(* Logix 5000 project; controller MetsoFilter vendor 1 type 14 code 106 rev 32.11; software revision 32.00; part 3 of 4 *)
(* tags used below, declared in another part *)
   AlarmHornPulser : BOOL;   // Pulse Horn during a new alarm
   AlarmReset : BOOL;   // Alarm Rest Relay
   ALM_W2 : DINT;   // Alarms to HMI, Word #2
   AlwaysOff : BOOL;   // Always Off Bit
   AS_AirDry : BOOL;   // Auto Sequence, Air Dry
   AS_ClothVibWash : BOOL;   // Auto Sequence Vibrate & Wash Cloth
   AS_ClothVibWash_T : TIMER;   // Auto Sequence Vibrate & Wash Cloth Timer
   AS_Drain : BOOL;   // Auto Sequence, Drain
   AS_HPC_Open_V1_T : TIMER;   // Auto Sequence, Open Slurry Valve V1 Timer
   AS_LowFeedWeight : BOOL;   // Auto Sequence, Low Feed Weight, Enable Retry
   AS_LowPressClose : BOOL;   // Auto Sequence, Close Press at Low Pressure
   AS_MembComp : BOOL;   // Auto Sequence, Membrane Compress
   AS_MembComp_Ena : BOOL;   // Auto Sequence, Enable Membrane Compress When in Auto Run
   AS_TopBlow_Wat : BOOL;   // Auto Sequence, Top Blow Water
   AS_TopBlowAir1 : BOOL;   // Auto Sequence, Top Blow Air #1
   AS_TopBlowAir1_T : TIMER;   // Auto Sequence, Top Blow Air #1 Timer
   AS_TopBlowAir2 : BOOL;   // Auto Sequence, Top Blow Air #2
   AS_TopBlowAir2_T : TIMER;   // Auto Sequence, Top Blow Air #2 Timer
   AS_VibrateCloth : BOOL;   // Auto Sequence Vibrate Cloth
   AS_VibrateCloth_T : TIMER;   // Auto Sequence Vibrate Cloth Timer
   Auto_Run : BOOL;   // Run the Next Step of the Auto Sequence
   AutoSeqStarted : BOOL;   // Auto Sequence Started
   ClothDamaged_T : TIMER;   // Dammaged Cloth Detection Switch On Plus Time
   Colon_STR : STRING;   // Constant Colon String = ":"
   Dash_STR : STRING;   // Constant Dash String = "-"
   DateTimeArray : DINT[7];
   Day_STR : STRING;   // Day String(1-31)
   DD_Cycle_1 : Status_Cycle;   // Cycle 1 At Left Side Of Statistics Screen
   DD_Cycle_2 : Status_Cycle;   // Cycle 2
   DD_Cycle_3 : Status_Cycle;   // Cycle 3
   DD_Cycle_4 : Status_Cycle;   // Cycle 4
   DD_Cycle_5 : Status_Cycle;   // Cycle 5
   DD_Cycle_6 : Status_Cycle;   // Cycle 6
   DD_Cycle_7_Now : Status_Cycle;   // Cycle 7, Now being Updated @ Right Side of Statistics Screen
   DD_CyclesLeft : DINT;   // To HMI, Cycles Left Before Servicing
   DD_CycleTime : DINT;   // To HMI, Current Cycle time
   DD_Date_STR : STRING;   // Date String - YYYY-MM-DD
   DD_Day_1 : Status_Day;   // Status Day 1 At Left Side of Statistics Screen
   DD_Day_2 : Status_Day;   // Status Day 2
   DD_Day_3 : Status_Day;   // Status Day 3
   DD_Day_4 : Status_Day;   // Status Day 4
   DD_Day_5 : Status_Day;   // Status Day 5
   DD_Day_6 : Status_Day;   // Status Day 6
   DD_Day_7_Now : Status_Day;   // Status Day 7, Now Being Updated @ Right Side of Statistics Screen
   DD_LastResetDate_STR : DINT;   // On Statistics Screen, Date when last reset performed
   DD_PressWeight : DINT;   // Press Weight from Analog Input Data Display
   DD_Shift3_Start : DINT;   // To HMI, Shift 3 Start Hour
   DD_Time_STR : STRING;   // Time String = HH:MM
   DD_TotalCycles : DINT;   // To HMI, Total Cycles Performed, since last Reset
   DD_TotalTons : DINT;   // To HMI, Total Tons Pressed from Last Reset
   DE_ServiceCycles : DINT;   // Special Screen, Service Cycles for Maintenance Data Entry
   DE_Shift1_Start : DINT;   // Special Screen, Shift1 Start Hour, Data Entry
   DE_Shift2_Start : DINT;   // Special Screen, Shift 2 Start Data Entry
   DSH1 : BOOL;   // Dammaged Cloth Detection Switch
   DummyOutput : BOOL;   // Dummy Output for Temporary outputs File
   GSC11 : BOOL;   // Upper Hatch is Closed Proximity Switch
   GSC9 : BOOL;   // Lower Hatch is Closed Proximity Switch
   GSO10 : BOOL;   // Lower Hatch is Open Proximity Switch
   GSO12 : BOOL;   // Upper Hatch is Open Proximity Switch
   H1b : BOOL;   // Hydraulic Valve, Main Drainage
   H2a : BOOL;   // Hydraulic Valve, High Pressure Drainage
   H2b : BOOL;   // Hydraulic Valve, High Pressure Close
   H3a : BOOL;   // Hydraulic Valve, Press Close
   H3b : BOOL;   // Hydraulic Valve, Press Open
   H4a : BOOL;   // Hydraulic Valve, Raise (Open) Lower Hatch
   H4b : BOOL;   // Hydraulic Valve, Lower (Close) Lower Hatch
   H5a : BOOL;   // Hydraulic Valve, Raise (Open) Upper Hatch
   H5b : BOOL;   // Hydraulic Valve, Lower (Close) Upper Hatch
   HornPulseDuration_T : TIMER;   // Pulse Horn Duration Timer
   HornPulseOff_T : TIMER;   // Pulse Horn Off Timer
   HornPulses_C : COUNTER;   // Number of times horn pusles for new alarm
   Hour_STR : STRING;   // Hour String(0-23)
   M_HPP_Run : BOOL;   // High Pressure Pump Run Output Bit
   M_HPP_Running : BOOL;   // High Pressure Pump is Running
   M_LPP_Run : BOOL;   // Low Pressure Pump Run Output Bit
   M_Vibrator_Run : BOOL;   // Vibrator Motor Run Output
   M_Vibrator_Run_T : TIMER;   // Vibrator Motor Run Output On Plus Time
   M_Vibrator_Running : BOOL;   // Vibrator Motor Running Input
   MAN_Vibrate : BOOL;   // Manual Vibrate Flip Flop
   Manual_ON : BOOL;   // Manual On Mode
   MAS_CloseHatch : BOOL;   // Manual / Auto Close Hatch
   MAS_CloseUpperHatch_T : TIMER;   // Manual / Auto Close Upper Hatch Delay Timer
   MAS_OpenHatch : BOOL;   // Manual / Auto Open Hatch
   MAS_OpenLowerHatch_T : TIMER;   // Manual / Auto Open Hatch, Delay Lower Hatch Open
   Minute_STR : STRING;   // Minute String(0-59)
   Month_STR : STRING;   // Month String(1-12)
   NewAlarm_OS : BOOL;   // A New Alarm Has Occured
   NewAlarm_PulseHorn : BOOL;   // A New Alarm has Occured, pulse the Horn
   NumberOfAlarms : DINT;   // Number of Active Alarms
   NumberOfAlarms_LS : DINT;   // Number of Active Alarms Last Scan, Detect New Alarm
   OneThirdAir1Preset : DINT;   // 1/3 Top Blow Air 1 time
   OneThirdAir2Preset : DINT;   // 1/3 Top Blow Air 2 time
   PB_AlarmAck : BOOL;   // Alarm Acknowledge Pushbutton
   PB_AlarmReset : BOOL;   // Alarm Reset Pushbutton
   PB_ResetSpecial : BOOL;   // Reset Pushbutton on the Specal Screen, Reset Total Cycles & Weight
   S_AS_DoneOS : BOOL;   // Statistics, Automatic Sequence Normally Done or Abnormally Stopped One Shot
   S_AS_DoneOSB : BOOL;   // Statistics, Automatic Sequence Done One Shot
   S_AS_StartOS : BOOL;   // Statistics, Automatic Sequence Started One Shot
   S_AS_StartOSB : BOOL;   // Statistics, Automatic Sequence Started One Shot
   S_CloseHatchOSB : BOOL;   // Statistics, Hatch Starting to Close, One Shot
   S_CycleTimer : TIMER;   // Statistics, Cycle Time Timer
   S_DryingTimer : TIMER;   // Statistics, Drying Time Timer
   S_NewDay : BOOL;   // Statistics, Midnight & No Sequence Running, Update Days
   S_OpenHatchOSB : BOOL;   // Statistics, Hatch Starting to Open, One Shot
   S_PressWeightTons : REAL;   // Statistics, Weight in Tons Just Pressed
   S_PumpTimer : TIMER;   // Statistics, Pump Time Timer
   S_Shift1 : BOOL;   // Statistics, Shift 1 in Progress
   S_Shift1_OSB : BOOL;   // Statistics, Start of Shift 1 One shot
   S_Shift2 : BOOL;   // Statistics, Shift 2 in Progress
   S_Shift2_OSB : BOOL;   // Statistics, Start of Shift 2 One shot
   S_Shift3 : BOOL;   // Statistics, Shift 3 in Progress
   S_Shift3_OSB : BOOL;   // Statistics, Start of Shift 3 One shot
   S_TempDINT : DINT;   // Statistics, Tempory Holding DINT
   S_WeightHatchOpen : DINT;   // Statistics, Weight of Press just as hatches Open
   S_ZeroHour_Latch : BOOL;   // Zero Hour Latch, wait for current sequence to finish, if running
   S_ZeroHour_OSB : BOOL;   // Hour = Zero, New Day One Shot
   TwoThirdsAir1Preset : DINT;   // 2/3 Top Blow Air 1 time
   TwoThirdsAir2Preset : DINT;   // 2/3 Top Blow Air 2 time
   Year_STR : STRING;   // Year String
   YV1 : BOOL;   // Valve #1, Slurry Supply, Open Output Bit
   YV10 : BOOL;   // Valve #10, Membrane Drain, Normally Open, Energize to Close, Output Bit
   YV3 : BOOL;   // Valve #3, Filtrate, Open Output Bit
   YV4 : BOOL;   // Valve #4, Slurry Return, Open Output Bit
   YV5 : BOOL;   // Valve #5, Drying Air, Open Output Bit
   YV6 : BOOL;   // Valve #6, Top Blow Air, Open Output Bit
   YV7 : BOOL;   // Valve #7, Membrane Air, Open Output Bit
   YV8 : BOOL;   // Valve #8, Top Blow Water, Open Output Bit
   YV9 : BOOL;   // Valve #9, Wash Water, Open Ouput Bit
   Zero_STR : STRING;   // Constant String= "0" Pad Values <10 0-9 -> 00-09
(* MainProgram, continued *)

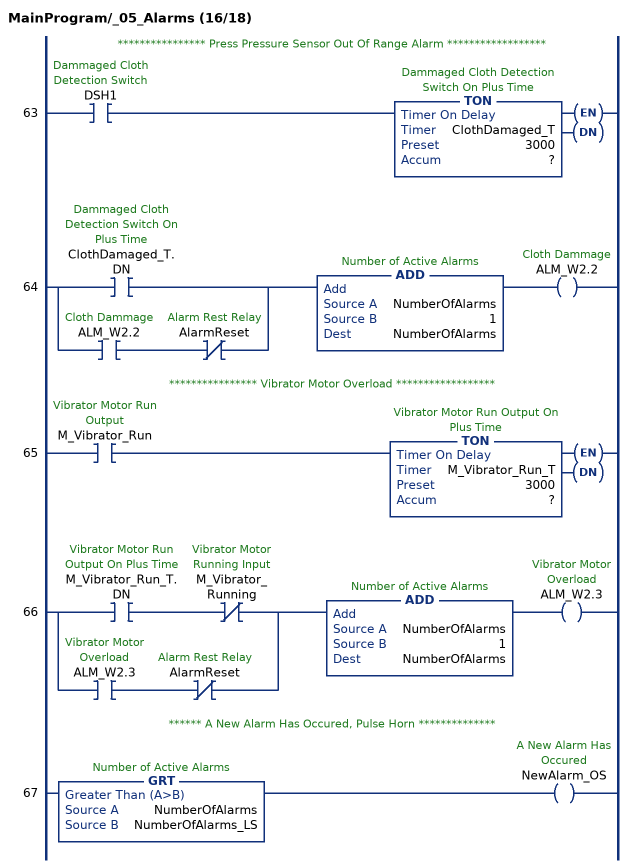
   [picture p48: MainProgram/_05_Alarms rungs 63-67]
   // **************** Press Pressure Sensor Out Of Range Alarm ******************
   63: XIC(DSH1)TON(ClothDamaged_T,?,?);
   64: [XIC(ClothDamaged_T.DN) ,XIC(ALM_W2.2) XIO(AlarmReset) ]ADD(NumberOfAlarms,1,NumberOfAlarms)OTE(ALM_W2.2);
   // **************** Vibrator Motor Overload ******************
   65: XIC(M_Vibrator_Run)TON(M_Vibrator_Run_T,?,?);
   66: [XIC(M_Vibrator_Run_T.DN) XIO(M_Vibrator_Running) ,XIC(ALM_W2.3) XIO(AlarmReset) ]ADD(NumberOfAlarms,1,NumberOfAlarms)OTE(ALM_W2.3);
   // ****** A New Alarm Has Occured, Pulse Horn **************
   67: GRT(NumberOfAlarms,NumberOfAlarms_LS)OTE(NewAlarm_OS);
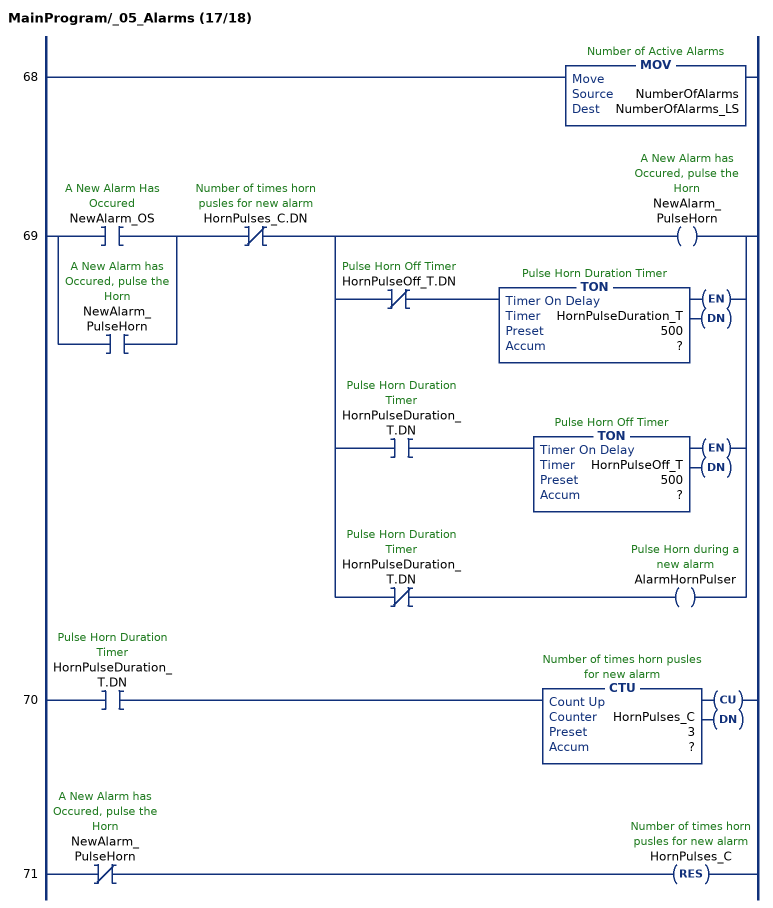
   68: MOV(NumberOfAlarms,NumberOfAlarms_LS);
   69: [XIC(NewAlarm_OS) ,XIC(NewAlarm_PulseHorn) ]XIO(HornPulses_C.DN)[OTE(NewAlarm_PulseHorn) ,XIO(HornPulseOff_T.DN) TON(HornPulseDuration_T,?,?) ,XIC(HornPulseDuration_T.DN) TON(HornPulseOff_T,?,?) ,XIO(HornPulseDuration_T.DN) OTE(AlarmHornPulser) ];
   70: XIC(HornPulseDuration_T.DN)CTU(HornPulses_C,?,?);
   71: XIO(NewAlarm_PulseHorn)RES(HornPulses_C);
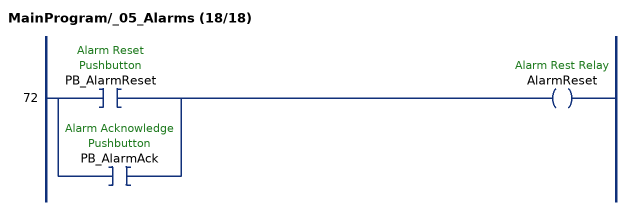
   72: [XIC(PB_AlarmReset) ,XIC(PB_AlarmAck) ]OTE(AlarmReset);
END_ROUTINE

ROUTINE _06_Output_Bits   (* ladder *)
// Set the Output Bits per Manual and Automatic Logic
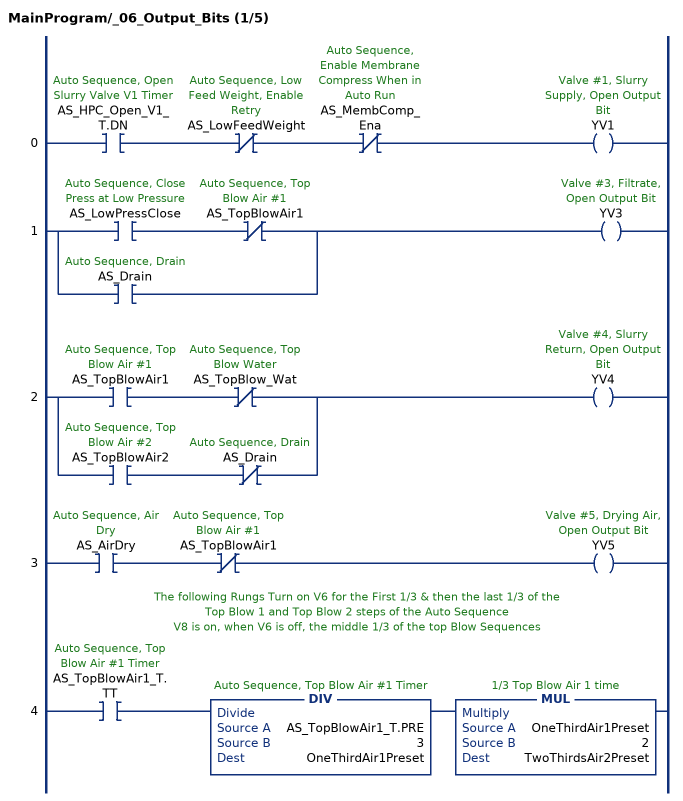
   0: XIC(AS_HPC_Open_V1_T.DN)XIO(AS_LowFeedWeight)XIO(AS_MembComp_Ena)OTE(YV1);
   1: [XIC(AS_LowPressClose) XIO(AS_TopBlowAir1) ,XIC(AS_Drain) ]OTE(YV3);
   2: [XIC(AS_TopBlowAir1) XIO(AS_TopBlow_Wat) ,XIC(AS_TopBlowAir2) XIO(AS_Drain) ]OTE(YV4);
   3: XIC(AS_AirDry)XIO(AS_TopBlowAir1)OTE(YV5);
   // The following Rungs Turn on V6 for the First 1/3 & then the last 1/3 of the
   // Top Blow 1 and Top Blow 2 steps of the Auto Sequence
   // V8 is on, when V6 is off, the middle 1/3 of the top Blow Sequences
   4: XIC(AS_TopBlowAir1_T.TT)DIV(AS_TopBlowAir1_T.PRE,3,OneThirdAir1Preset)MUL(OneThirdAir1Preset,2,TwoThirdsAir2Preset);
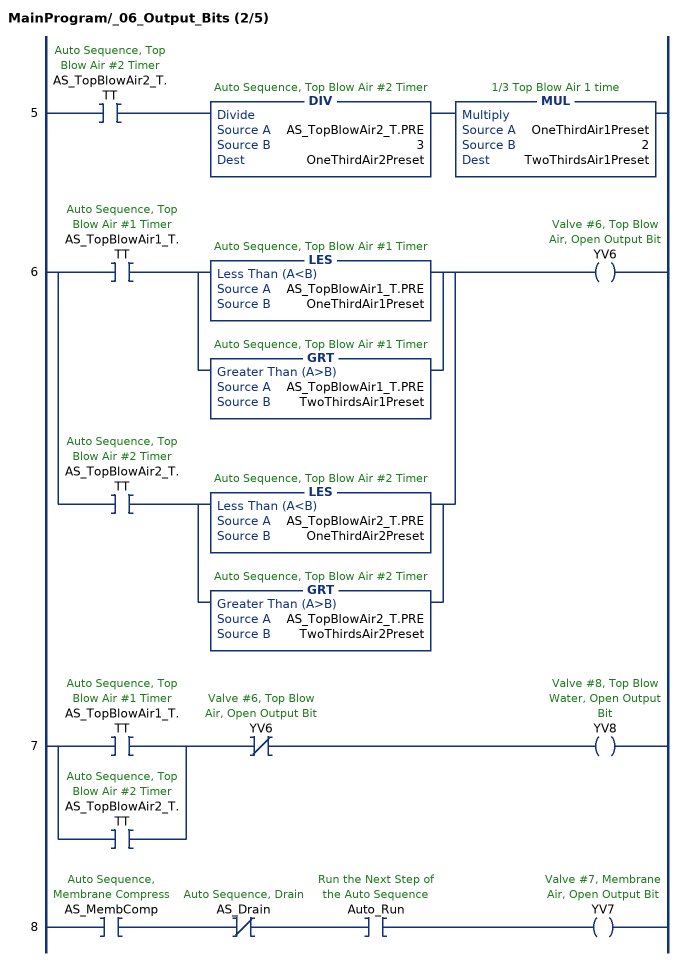
   5: XIC(AS_TopBlowAir2_T.TT)DIV(AS_TopBlowAir2_T.PRE,3,OneThirdAir2Preset)MUL(OneThirdAir1Preset,2,TwoThirdsAir1Preset);
   6: [XIC(AS_TopBlowAir1_T.TT) [LES(AS_TopBlowAir1_T.PRE,OneThirdAir1Preset) ,GRT(AS_TopBlowAir1_T.PRE,TwoThirdsAir1Preset) ] ,XIC(AS_TopBlowAir2_T.TT) [LES(AS_TopBlowAir2_T.PRE,OneThirdAir2Preset) ,GRT(AS_TopBlowAir2_T.PRE,TwoThirdsAir2Preset) ] ]OTE(YV6);
   7: [XIC(AS_TopBlowAir1_T.TT) ,XIC(AS_TopBlowAir2_T.TT) ]XIO(YV6)OTE(YV8);
   8: XIC(AS_MembComp)XIO(AS_Drain)XIC(Auto_Run)OTE(YV7);
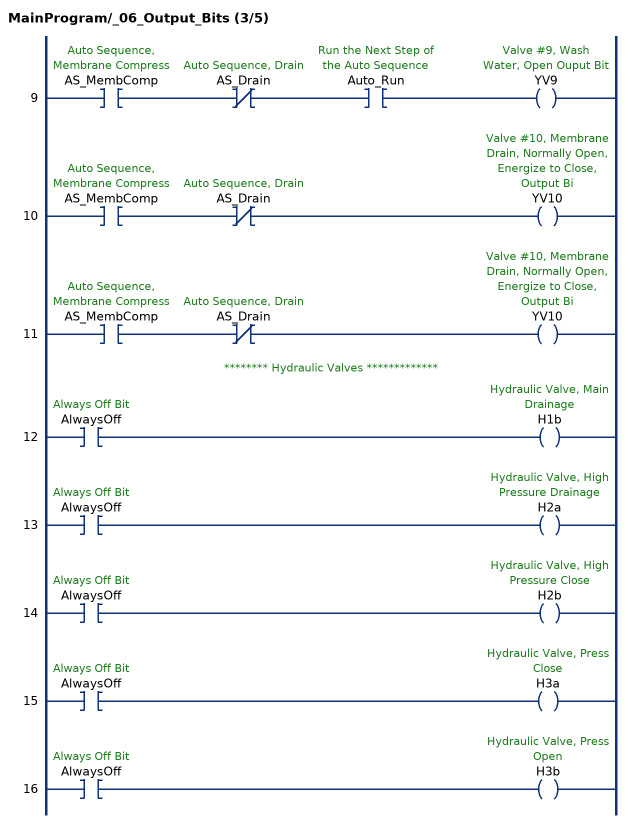
   9: XIC(AS_MembComp)XIO(AS_Drain)XIC(Auto_Run)OTE(YV9);
   10: XIC(AS_MembComp)XIO(AS_Drain)OTE(YV10);
   11: XIC(AS_MembComp)XIO(AS_Drain)OTE(YV10);
   // ******** Hydraulic Valves *************
   12: XIC(AlwaysOff)OTE(H1b);
   13: XIC(AlwaysOff)OTE(H2a);
   14: XIC(AlwaysOff)OTE(H2b);
   15: XIC(AlwaysOff)OTE(H3a);
   16: XIC(AlwaysOff)OTE(H3b);
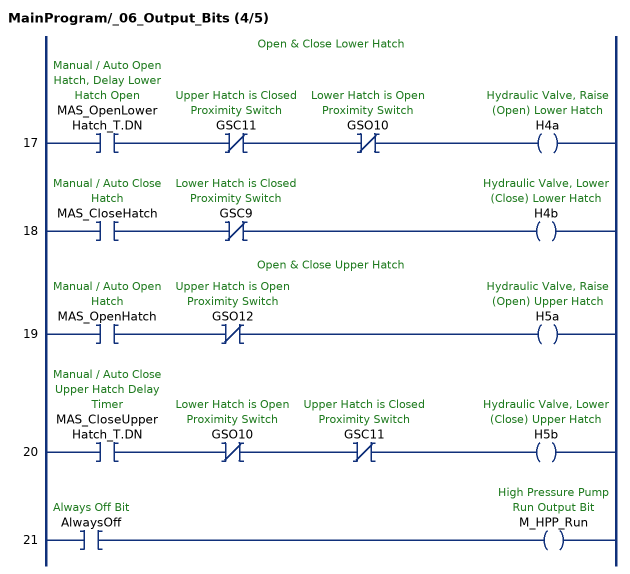
   // Open & Close Lower Hatch
   17: XIC(MAS_OpenLowerHatch_T.DN)XIO(GSC11)XIO(GSO10)OTE(H4a);
   18: XIC(MAS_CloseHatch)XIO(GSC9)OTE(H4b);
   // Open & Close Upper Hatch
   19: XIC(MAS_OpenHatch)XIO(GSO12)OTE(H5a);
   20: XIC(MAS_CloseUpperHatch_T.DN)XIO(GSO10)XIO(GSC11)OTE(H5b);
   21: XIC(AlwaysOff)OTE(M_HPP_Run);
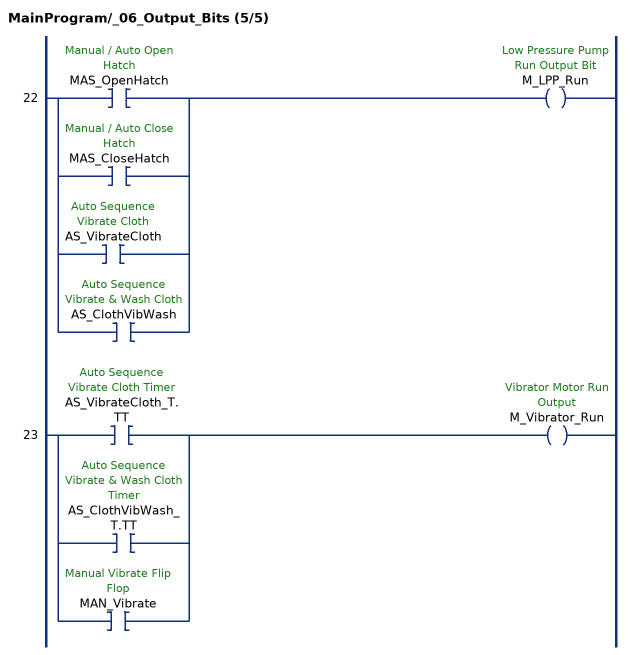
   22: [XIC(MAS_OpenHatch) ,XIC(MAS_CloseHatch) ,XIC(AS_VibrateCloth) ,XIC(AS_ClothVibWash) ]OTE(M_LPP_Run);
   23: [XIC(AS_VibrateCloth_T.TT) ,XIC(AS_ClothVibWash_T.TT) ,XIC(MAN_Vibrate) ]OTE(M_Vibrator_Run);
END_ROUTINE

ROUTINE _07_MapOutputs   (* ladder *)
// Map Output Bits to PLC Outputs
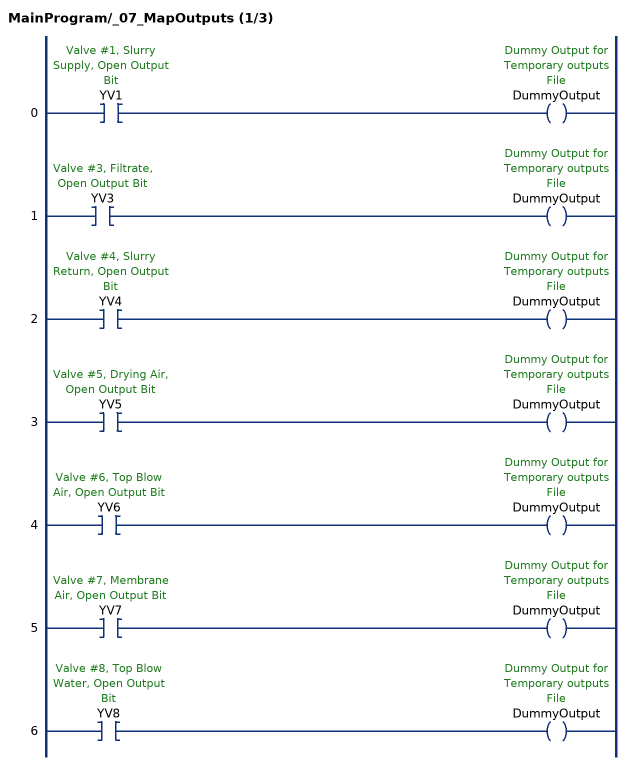
   0: XIC(YV1)OTE(DummyOutput);
   1: XIC(YV3)OTE(DummyOutput);
   2: XIC(YV4)OTE(DummyOutput);
   3: XIC(YV5)OTE(DummyOutput);
   4: XIC(YV6)OTE(DummyOutput);
   5: XIC(YV7)OTE(DummyOutput);
   6: XIC(YV8)OTE(DummyOutput);
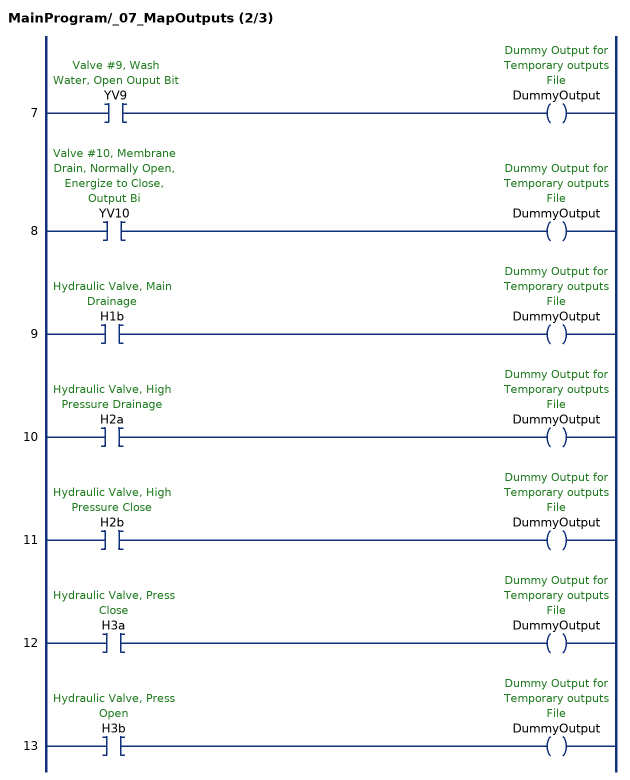
   7: XIC(YV9)OTE(DummyOutput);
   8: XIC(YV10)OTE(DummyOutput);
   9: XIC(H1b)OTE(DummyOutput);
   10: XIC(H2a)OTE(DummyOutput);
   11: XIC(H2b)OTE(DummyOutput);
   12: XIC(H3a)OTE(DummyOutput);
   13: XIC(H3b)OTE(DummyOutput);
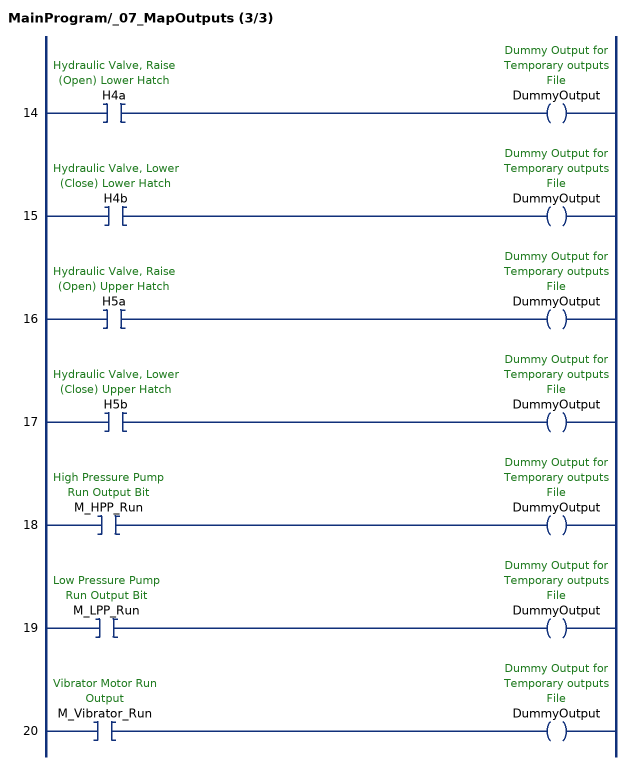
   14: XIC(H4a)OTE(DummyOutput);
   15: XIC(H4b)OTE(DummyOutput);
   16: XIC(H5a)OTE(DummyOutput);
   17: XIC(H5b)OTE(DummyOutput);
   18: XIC(M_HPP_Run)OTE(DummyOutput);
   19: XIC(M_LPP_Run)OTE(DummyOutput);
   20: XIC(M_Vibrator_Run)OTE(DummyOutput);
END_ROUTINE

ROUTINE _08_Statistics   (* ladder *)
// Track Last 7 Days & Cycles
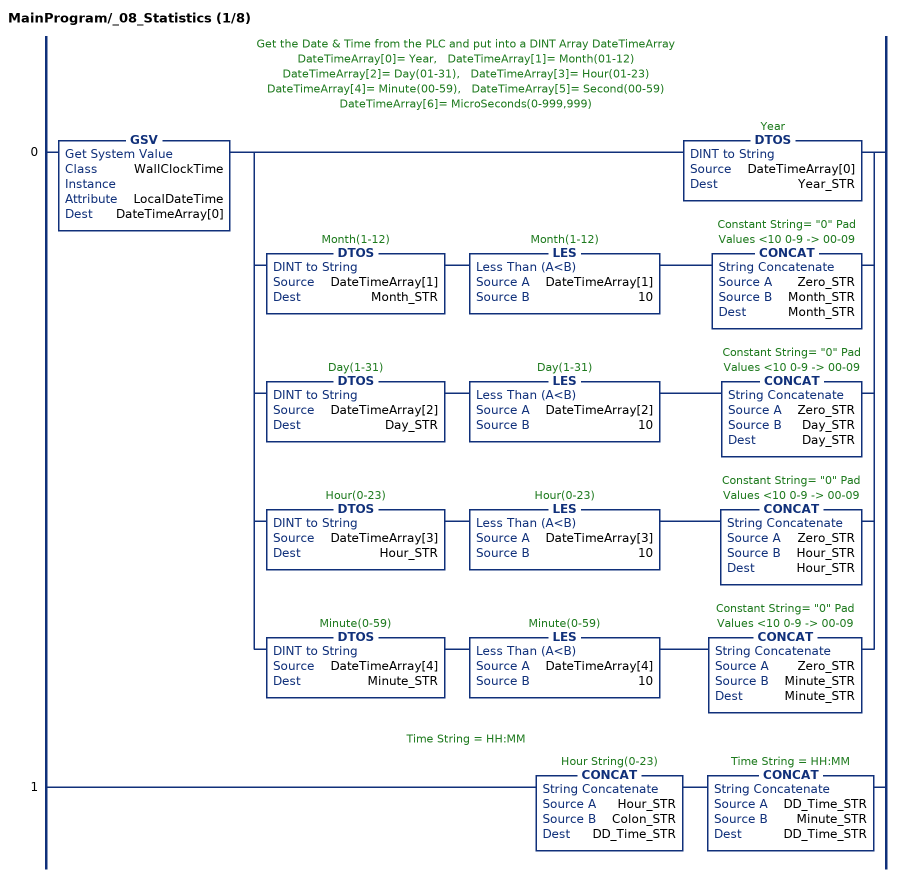
   // Get the Date & Time from the PLC and put into a DINT Array DateTimeArray
   // DateTimeArray[0]= Year,   DateTimeArray[1]= Month(01-12)
   // DateTimeArray[2]= Day(01-31),   DateTimeArray[3]= Hour(01-23)
   // DateTimeArray[4]= Minute(00-59),   DateTimeArray[5]= Second(00-59)
   // DateTimeArray[6]= MicroSeconds(0-999,999)
   0: GSV(WallClockTime,,LocalDateTime,DateTimeArray[0])[DTOS(DateTimeArray[0],Year_STR) ,DTOS(DateTimeArray[1],Month_STR) LES(DateTimeArray[1],10) CONCAT(Zero_STR,Month_STR,Month_STR) ,DTOS(DateTimeArray[2],Day_STR) LES(DateTimeArray[2],10) CONCAT(Zero_STR,Day_STR,Day_STR) ,DTOS(DateTimeArray[3],Hour_STR) LES(DateTimeArray[3],10) CONCAT(Zero_STR,Hour_STR,Hour_STR) ,DTOS(DateTimeArray[4],Minute_STR) LES(DateTimeArray[4],10) CONCAT(Zero_STR,Minute_STR,Minute_STR) ];
   // Time String = HH:MM
   1: CONCAT(Hour_STR,Colon_STR,DD_Time_STR)CONCAT(DD_Time_STR,Minute_STR,DD_Time_STR);
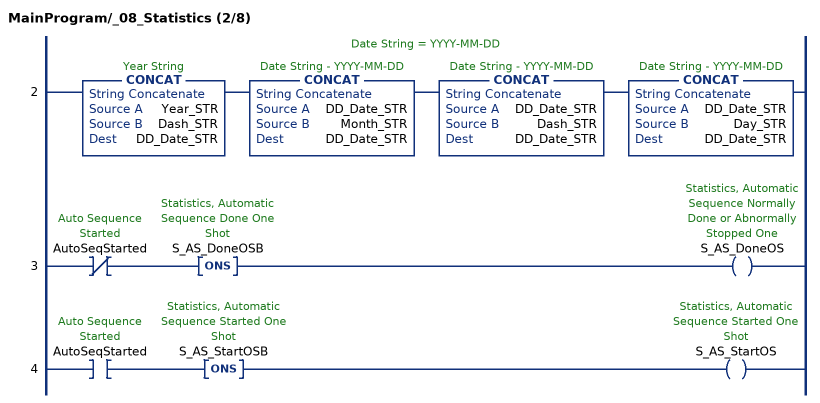
   // Date String = YYYY-MM-DD
   2: CONCAT(Year_STR,Dash_STR,DD_Date_STR)CONCAT(DD_Date_STR,Month_STR,DD_Date_STR)CONCAT(DD_Date_STR,Dash_STR,DD_Date_STR)CONCAT(DD_Date_STR,Day_STR,DD_Date_STR);
   3: XIO(AutoSeqStarted)ONS(S_AS_DoneOSB)OTE(S_AS_DoneOS);
   4: XIC(AutoSeqStarted)ONS(S_AS_StartOSB)OTE(S_AS_StartOS);
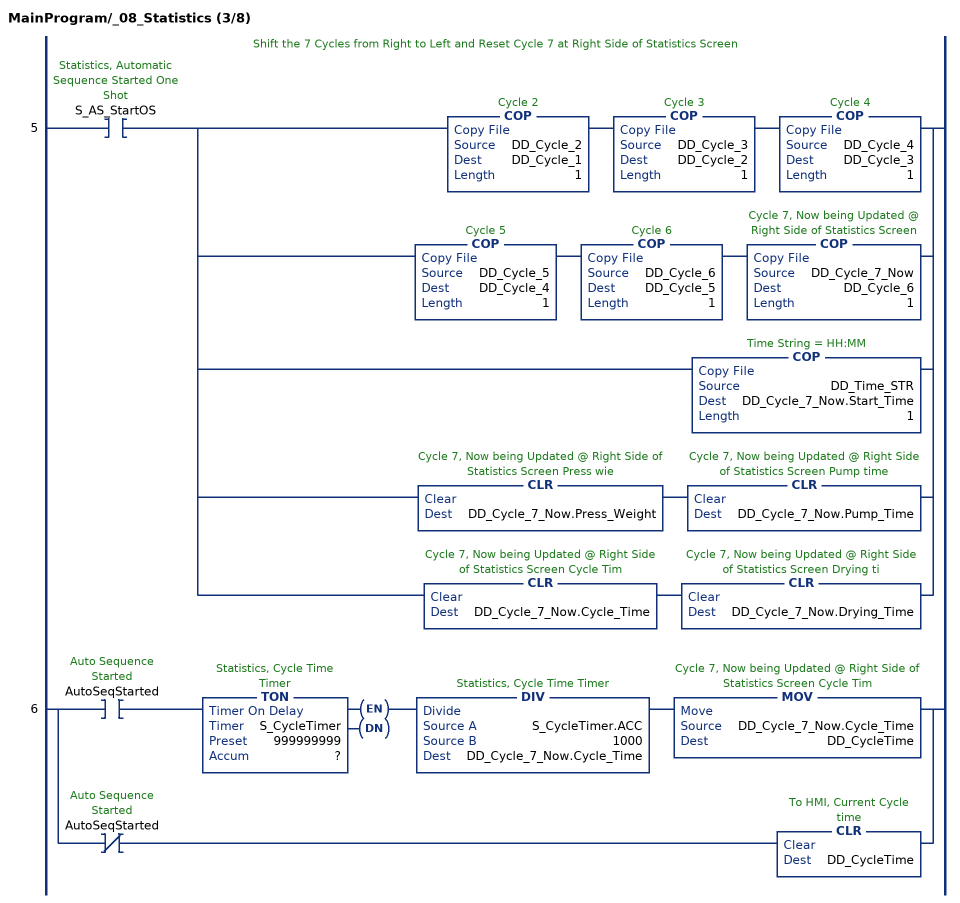
   // Shift the 7 Cycles from Right to Left and Reset Cycle 7 at Right Side of Statistics Screen
   5: XIC(S_AS_StartOS)[COP(DD_Cycle_2,DD_Cycle_1,1) COP(DD_Cycle_3,DD_Cycle_2,1) COP(DD_Cycle_4,DD_Cycle_3,1) ,COP(DD_Cycle_5,DD_Cycle_4,1) COP(DD_Cycle_6,DD_Cycle_5,1) COP(DD_Cycle_7_Now,DD_Cycle_6,1) ,COP(DD_Time_STR,DD_Cycle_7_Now.Start_Time,1) ,CLR(DD_Cycle_7_Now.Press_Weight) CLR(DD_Cycle_7_Now.Pump_Time) ,CLR(DD_Cycle_7_Now.Cycle_Time) CLR(DD_Cycle_7_Now.Drying_Time) ];
   6: [XIC(AutoSeqStarted) TON(S_CycleTimer,?,?) DIV(S_CycleTimer.ACC,1000,DD_Cycle_7_Now.Cycle_Time) MOV(DD_Cycle_7_Now.Cycle_Time,DD_CycleTime) ,XIO(AutoSeqStarted) CLR(DD_CycleTime) ];
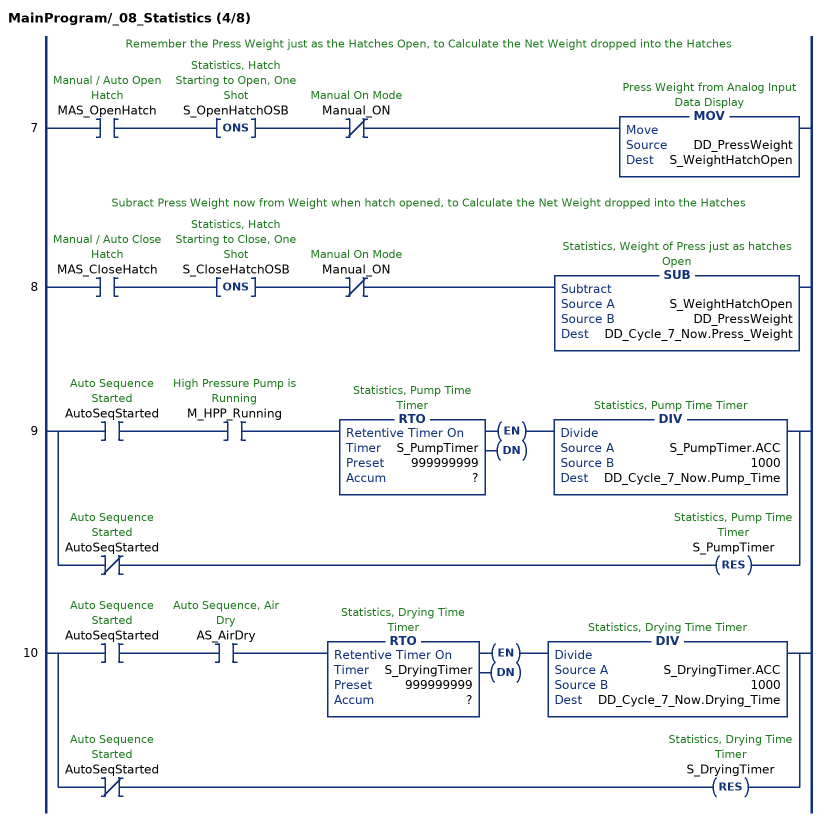
   // Remember the Press Weight just as the Hatches Open, to Calculate the Net Weight dropped into the Hatches
   7: XIC(MAS_OpenHatch)ONS(S_OpenHatchOSB)XIO(Manual_ON)MOV(DD_PressWeight,S_WeightHatchOpen);
   // Subract Press Weight now from Weight when hatch opened, to Calculate the Net Weight dropped into the Hatches
   8: XIC(MAS_CloseHatch)ONS(S_CloseHatchOSB)XIO(Manual_ON)SUB(S_WeightHatchOpen,DD_PressWeight,DD_Cycle_7_Now.Press_Weight);
   9: [XIC(AutoSeqStarted) XIC(M_HPP_Running) RTO(S_PumpTimer,?,?) DIV(S_PumpTimer.ACC,1000,DD_Cycle_7_Now.Pump_Time) ,XIO(AutoSeqStarted) RES(S_PumpTimer) ];
   10: [XIC(AutoSeqStarted) XIC(AS_AirDry) RTO(S_DryingTimer,?,?) DIV(S_DryingTimer.ACC,1000,DD_Cycle_7_Now.Drying_Time) ,XIO(AutoSeqStarted) RES(S_DryingTimer) ];
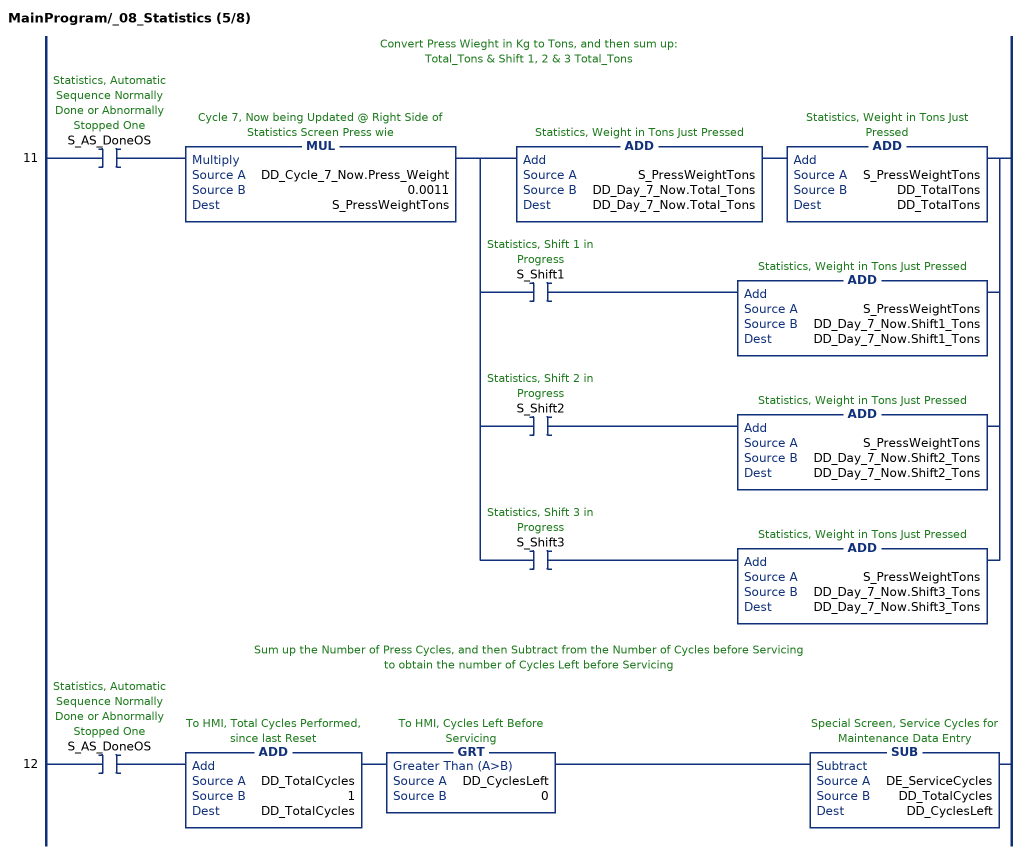
   // Convert Press Wieght in Kg to Tons, and then sum up:
   // Total_Tons & Shift 1, 2 & 3 Total_Tons
   11: XIC(S_AS_DoneOS)MUL(DD_Cycle_7_Now.Press_Weight,0.0011,S_PressWeightTons)[ADD(S_PressWeightTons,DD_Day_7_Now.Total_Tons,DD_Day_7_Now.Total_Tons) ADD(S_PressWeightTons,DD_TotalTons,DD_TotalTons) ,XIC(S_Shift1) ADD(S_PressWeightTons,DD_Day_7_Now.Shift1_Tons,DD_Day_7_Now.Shift1_Tons) ,XIC(S_Shift2) ADD(S_PressWeightTons,DD_Day_7_Now.Shift2_Tons,DD_Day_7_Now.Shift2_Tons) ,XIC(S_Shift3) ADD(S_PressWeightTons,DD_Day_7_Now.Shift3_Tons,DD_Day_7_Now.Shift3_Tons) ];
   // Sum up the Number of Press Cycles, and then Subtract from the Number of Cycles before Servicing
   // to obtain the number of Cycles Left before Servicing
   12: XIC(S_AS_DoneOS)ADD(DD_TotalCycles,1,DD_TotalCycles)GRT(DD_CyclesLeft,0)SUB(DE_ServiceCycles,DD_TotalCycles,DD_CyclesLeft);
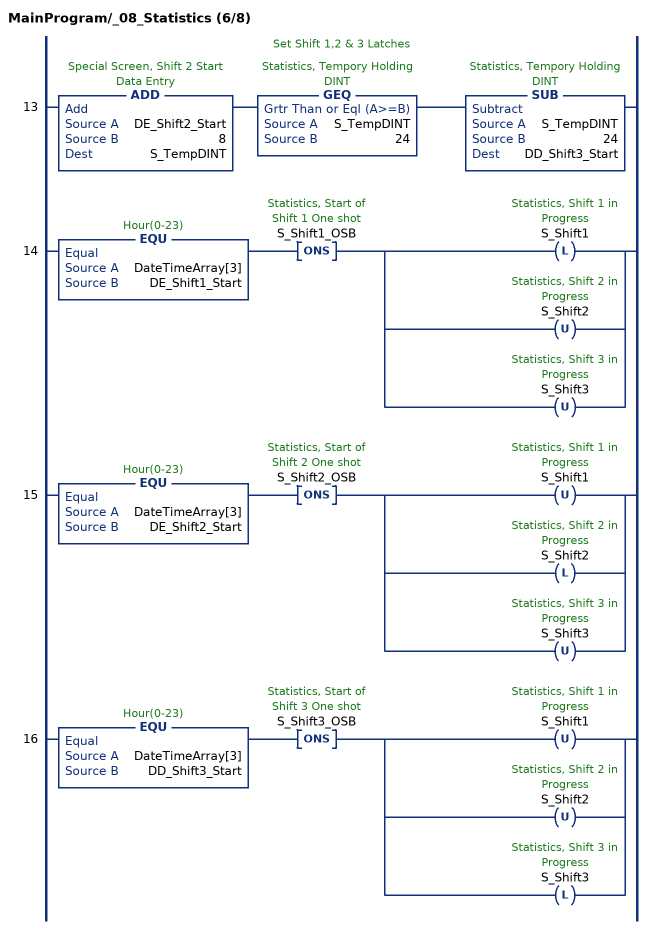
   // Set Shift 1,2 & 3 Latches
   13: ADD(DE_Shift2_Start,8,S_TempDINT)GEQ(S_TempDINT,24)SUB(S_TempDINT,24,DD_Shift3_Start);
   14: EQU(DateTimeArray[3],DE_Shift1_Start)ONS(S_Shift1_OSB)[OTL(S_Shift1) ,OTU(S_Shift2) ,OTU(S_Shift3) ];
   15: EQU(DateTimeArray[3],DE_Shift2_Start)ONS(S_Shift2_OSB)[OTU(S_Shift1) ,OTL(S_Shift2) ,OTU(S_Shift3) ];
   16: EQU(DateTimeArray[3],DD_Shift3_Start)ONS(S_Shift3_OSB)[OTU(S_Shift1) ,OTU(S_Shift2) ,OTL(S_Shift3) ];
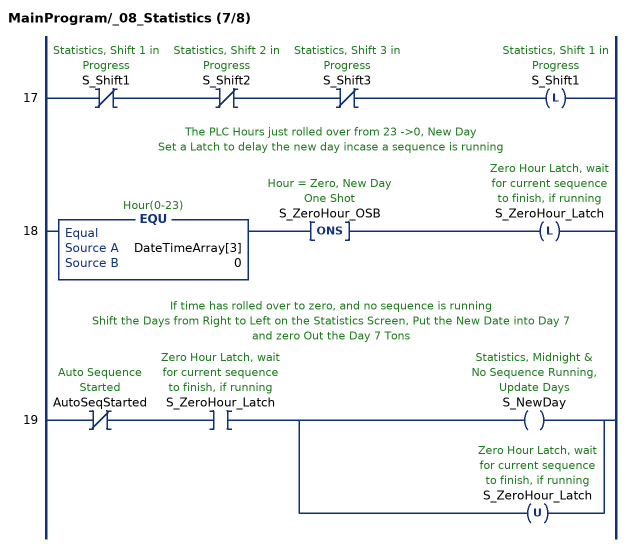
   17: XIO(S_Shift1)XIO(S_Shift2)XIO(S_Shift3)OTL(S_Shift1);
   // The PLC Hours just rolled over from 23 ->0, New Day
   // Set a Latch to delay the new day incase a sequence is running
   18: EQU(DateTimeArray[3],0)ONS(S_ZeroHour_OSB)OTL(S_ZeroHour_Latch);
   // If time has rolled over to zero, and no sequence is running
   // Shift the Days from Right to Left on the Statistics Screen, Put the New Date into Day 7
   // and zero Out the Day 7 Tons
   19: XIO(AutoSeqStarted)XIC(S_ZeroHour_Latch)[OTE(S_NewDay) ,OTU(S_ZeroHour_Latch) ];
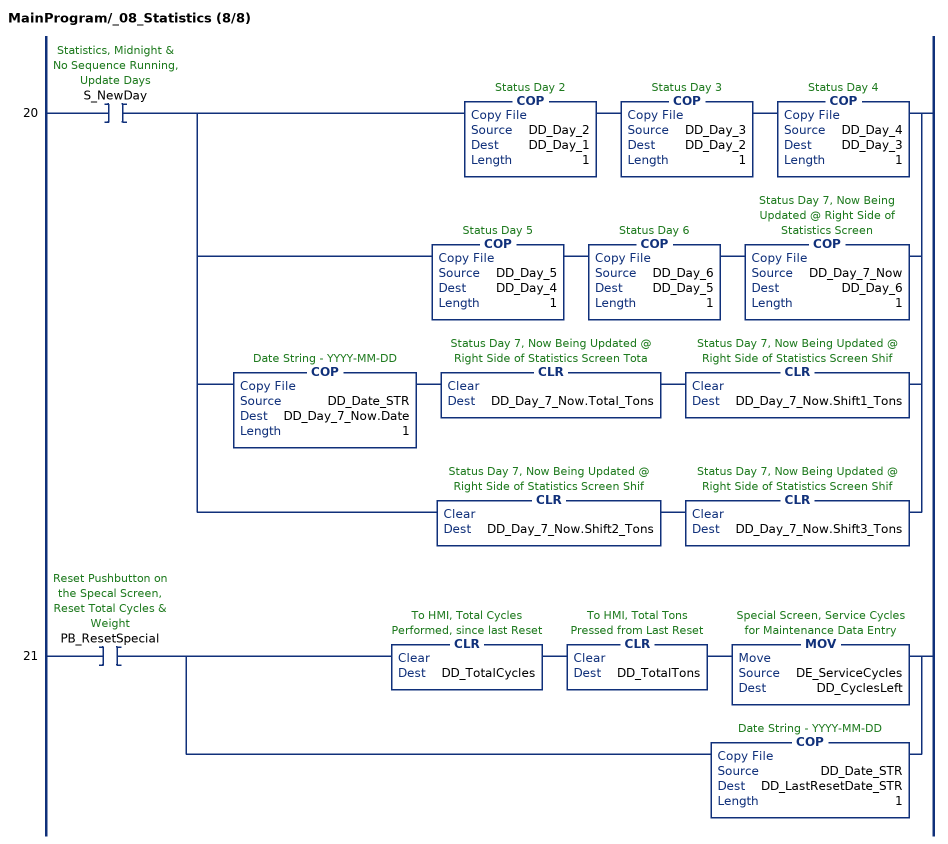
   20: XIC(S_NewDay)[COP(DD_Day_2,DD_Day_1,1) COP(DD_Day_3,DD_Day_2,1) COP(DD_Day_4,DD_Day_3,1) ,COP(DD_Day_5,DD_Day_4,1) COP(DD_Day_6,DD_Day_5,1) COP(DD_Day_7_Now,DD_Day_6,1) ,COP(DD_Date_STR,DD_Day_7_Now.Date,1) CLR(DD_Day_7_Now.Total_Tons) CLR(DD_Day_7_Now.Shift1_Tons) ,CLR(DD_Day_7_Now.Shift2_Tons) CLR(DD_Day_7_Now.Shift3_Tons) ];
   21: XIC(PB_ResetSpecial)[CLR(DD_TotalCycles) CLR(DD_TotalTons) MOV(DE_ServiceCycles,DD_CyclesLeft) ,COP(DD_Date_STR,DD_LastResetDate_STR,1) ];
END_ROUTINE
